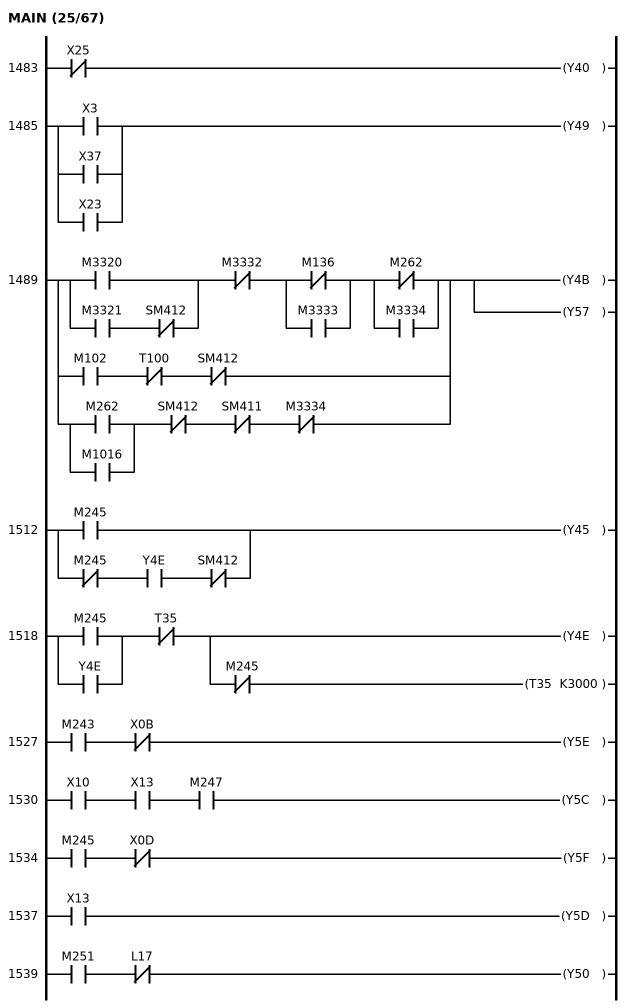
[picture p24: ladder of MAIN, rungs at steps 1483 to 1539]
1483  LDI     X25
      OUT     Y40
1485  LD      X3
      OR      X37
      OR      X23
      OUT     Y49
1489  LD      M3320
      LD      M3321
      ANI     SM412
      ORB
      ANI     M3332
      LDI     M136
      OR      M3333
      ANB
      LDI     M262
      OR      M3334
      ANB
      LD      M102
      ANI     T100
      ANI     SM412
      ORB
      LD      M262
      OR      M1016
      ANI     SM412
      ANI     SM411
      ANI     M3334
      ORB
      OUT     Y4B
      OUT     Y57
1512  LD      M245
      LDI     M245
      AND     Y4E
      ANI     SM412
      ORB
      OUT     Y45
1518  LD      M245
      OR      Y4E
      ANI     T35
      OUT     Y4E
      ANI     M245
      OUT     T35 K3000
1527  LD      M243
      ANI     X0B
      OUT     Y5E
1530  LD      X10
      AND     X13
      AND     M247
      OUT     Y5C
1534  LD      M245
      ANI     X0D
      OUT     Y5F
1537  LD      X13
      OUT     Y5D
1539  LD      M251
      ANI     L17
      OUT     Y50
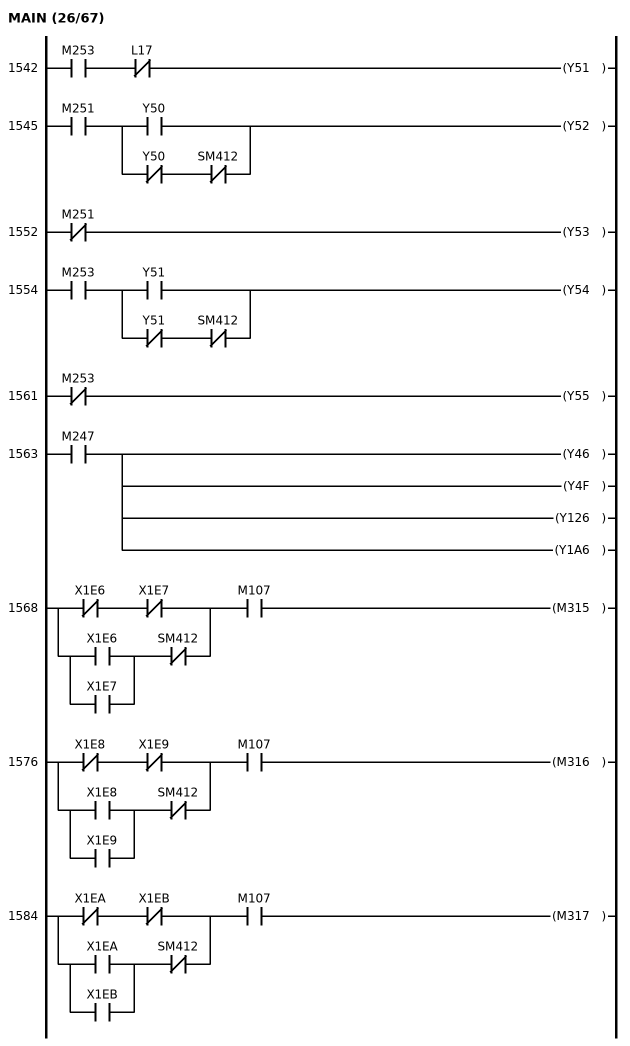
1542  LD      M253
      ANI     L17
      OUT     Y51
1545  LD      M251
      LD      Y50
      LDI     Y50
      ANI     SM412
      ORB
      ANB
      OUT     Y52
1552  LDI     M251
      OUT     Y53
1554  LD      M253
      LD      Y51
      LDI     Y51
      ANI     SM412
      ORB
      ANB
      OUT     Y54
1561  LDI     M253
      OUT     Y55
1563  LD      M247
      OUT     Y46
      OUT     Y4F
      OUT     Y126
      OUT     Y1A6
1568  LDI     X1E6
      ANI     X1E7
      LD      X1E6
      OR      X1E7
      ANI     SM412
      ORB
      AND     M107
      OUT     M315
1576  LDI     X1E8
      ANI     X1E9
      LD      X1E8
      OR      X1E9
      ANI     SM412
      ORB
      AND     M107
      OUT     M316
1584  LDI     X1EA
      ANI     X1EB
      LD      X1EA
      OR      X1EB
      ANI     SM412
      ORB
      AND     M107
      OUT     M317
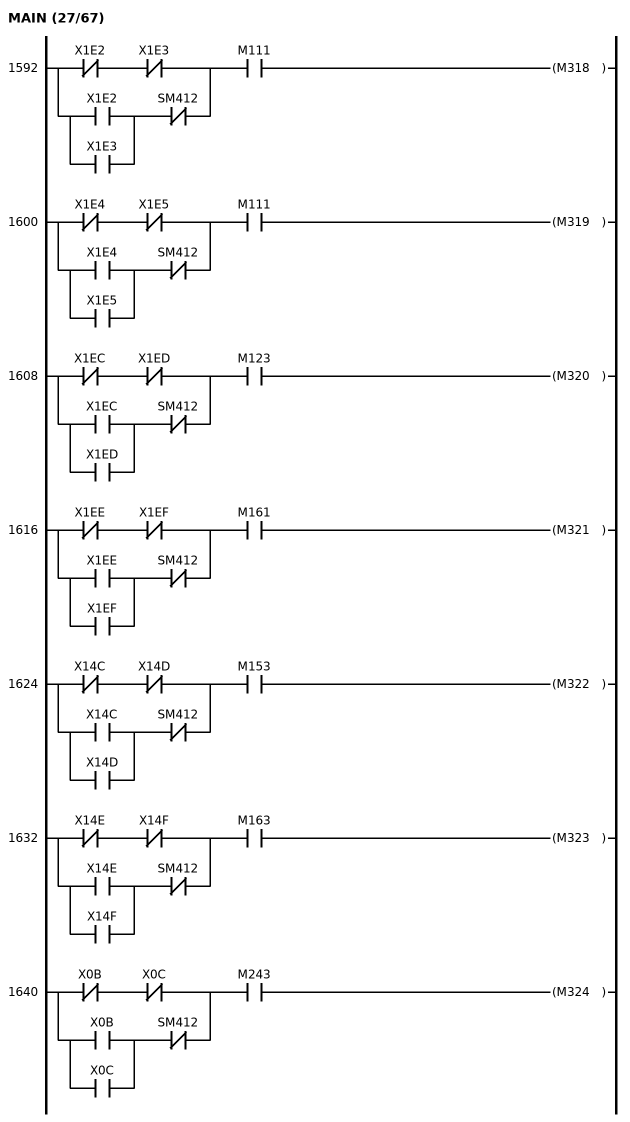
1592  LDI     X1E2
      ANI     X1E3
      LD      X1E2
      OR      X1E3
      ANI     SM412
      ORB
      AND     M111
      OUT     M318
1600  LDI     X1E4
      ANI     X1E5
      LD      X1E4
      OR      X1E5
      ANI     SM412
      ORB
      AND     M111
      OUT     M319
1608  LDI     X1EC
      ANI     X1ED
      LD      X1EC
      OR      X1ED
      ANI     SM412
      ORB
      AND     M123
      OUT     M320
1616  LDI     X1EE
      ANI     X1EF
      LD      X1EE
      OR      X1EF
      ANI     SM412
      ORB
      AND     M161
      OUT     M321
1624  LDI     X14C
      ANI     X14D
      LD      X14C
      OR      X14D
      ANI     SM412
      ORB
      AND     M153
      OUT     M322
1632  LDI     X14E
      ANI     X14F
      LD      X14E
      OR      X14F
      ANI     SM412
      ORB
      AND     M163
      OUT     M323
1640  LDI     X0B
      ANI     X0C
      LD      X0B
      OR      X0C
      ANI     SM412
      ORB
      AND     M243
      OUT     M324
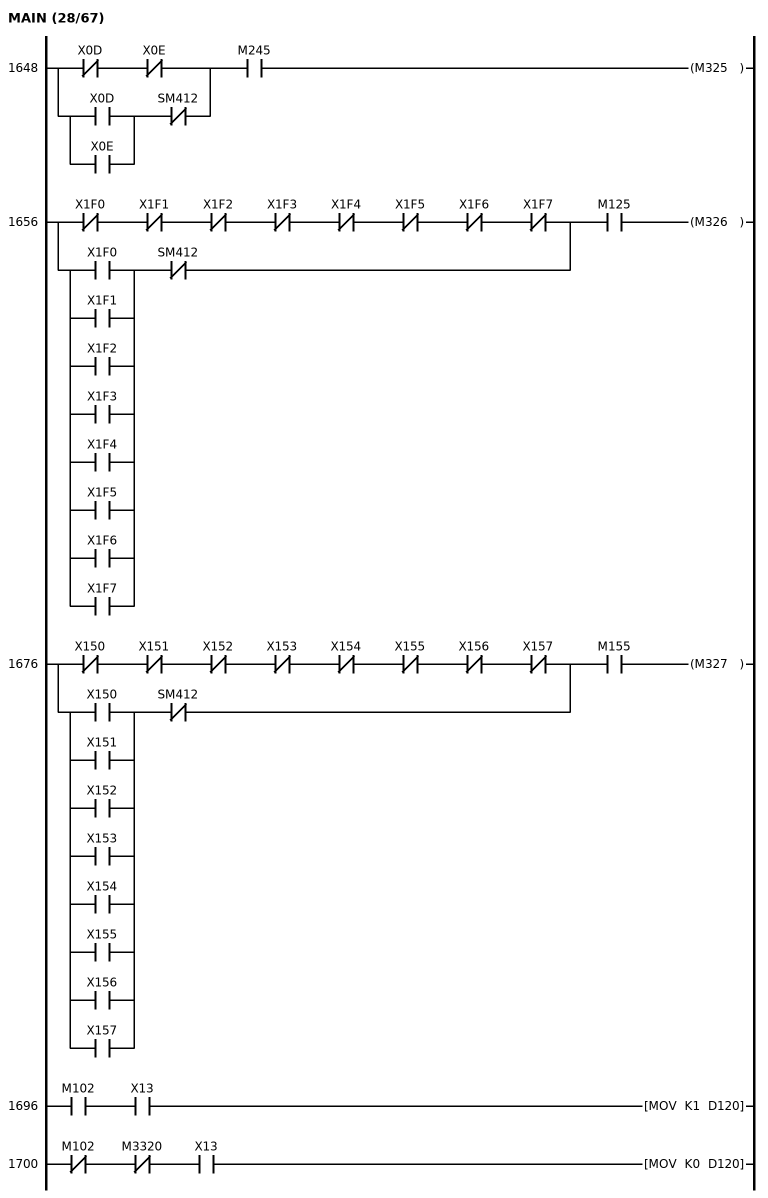
1648  LDI     X0D
      ANI     X0E
      LD      X0D
      OR      X0E
      ANI     SM412
      ORB
      AND     M245
      OUT     M325
1656  LDI     X1F0
      ANI     X1F1
      ANI     X1F2
      ANI     X1F3
      ANI     X1F4
      ANI     X1F5
      ANI     X1F6
      ANI     X1F7
      LD      X1F0
      OR      X1F1
      OR      X1F2
      OR      X1F3
      OR      X1F4
      OR      X1F5
      OR      X1F6
      OR      X1F7
      ANI     SM412
      ORB
      AND     M125
      OUT     M326
1676  LDI     X150
      ANI     X151
      ANI     X152
      ANI     X153
      ANI     X154
      ANI     X155
      ANI     X156
      ANI     X157
      LD      X150
      OR      X151
      OR      X152
      OR      X153
      OR      X154
      OR      X155
      OR      X156
      OR      X157
      ANI     SM412
      ORB
      AND     M155
      OUT     M327
1696  LD      M102
      AND     X13
      MOV     K1 D120
1700  LDI     M102
      ANI     M3320
      AND     X13
      MOV     K0 D120
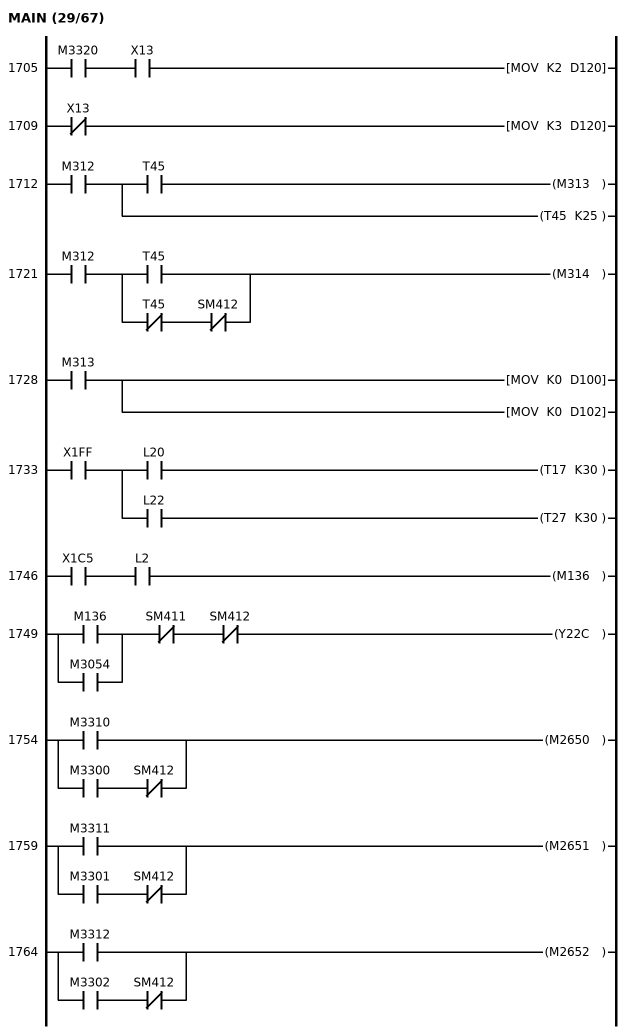
1705  LD      M3320
      AND     X13
      MOV     K2 D120
1709  LDI     X13
      MOV     K3 D120
1712  LD      M312
      MPS
      AND     T45
      OUT     M313
      MPP
      OUT     T45 K25
1721  LD      M312
      LD      T45
      LDI     T45
      ANI     SM412
      ORB
      ANB
      OUT     M314
1728  LD      M313
      MOV     K0 D100
      MOV     K0 D102
1733  LD      X1FF
      MPS
      AND     L20
      OUT     T17 K30
      MPP
      AND     L22
      OUT     T27 K30
1746  LD      X1C5
      AND     L2
      OUT     M136
1749  LD      M136
      OR      M3054
      ANI     SM411
      ANI     SM412
      OUT     Y22C
1754  LD      M3310
      LD      M3300
      ANI     SM412
      ORB
      OUT     M2650
1759  LD      M3311
      LD      M3301
      ANI     SM412
      ORB
      OUT     M2651
1764  LD      M3312
      LD      M3302
      ANI     SM412
      ORB
      OUT     M2652
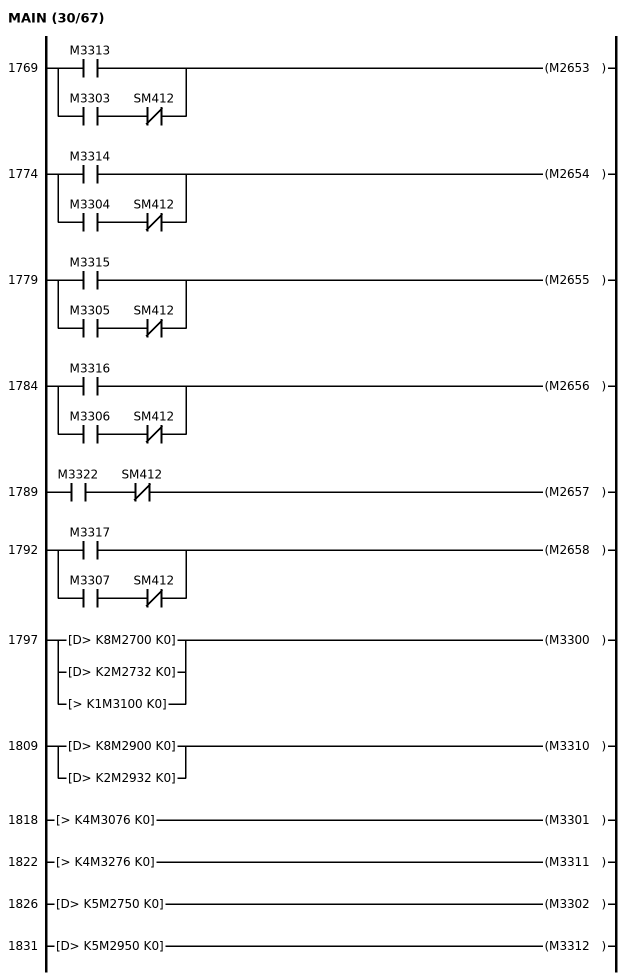
1769  LD      M3313
      LD      M3303
      ANI     SM412
      ORB
      OUT     M2653
1774  LD      M3314
      LD      M3304
      ANI     SM412
      ORB
      OUT     M2654
1779  LD      M3315
      LD      M3305
      ANI     SM412
      ORB
      OUT     M2655
1784  LD      M3316
      LD      M3306
      ANI     SM412
      ORB
      OUT     M2656
1789  LD      M3322
      ANI     SM412
      OUT     M2657
1792  LD      M3317
      LD      M3307
      ANI     SM412
      ORB
      OUT     M2658
1797  LDD>    K8M2700 K0
      ORD>    K2M2732 K0
      OR>     K1M3100 K0
      OUT     M3300
1809  LDD>    K8M2900 K0
      ORD>    K2M2932 K0
      OUT     M3310
1818  LD>     K4M3076 K0
      OUT     M3301
1822  LD>     K4M3276 K0
      OUT     M3311
1826  LDD>    K5M2750 K0
      OUT     M3302
1831  LDD>    K5M2950 K0
      OUT     M3312
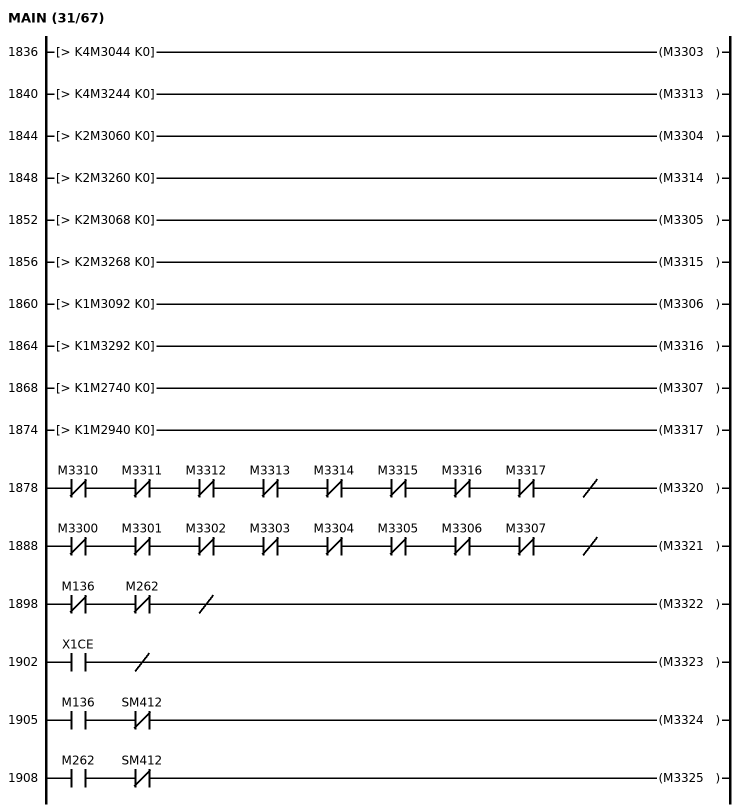
1836  LD>     K4M3044 K0
      OUT     M3303
1840  LD>     K4M3244 K0
      OUT     M3313
1844  LD>     K2M3060 K0
      OUT     M3304
1848  LD>     K2M3260 K0
      OUT     M3314
1852  LD>     K2M3068 K0
      OUT     M3305
1856  LD>     K2M3268 K0
      OUT     M3315
1860  LD>     K1M3092 K0
      OUT     M3306
1864  LD>     K1M3292 K0
      OUT     M3316
1868  LD>     K1M2740 K0
      OUT     M3307
        [note] 
1874  LD>     K1M2940 K0
      OUT     M3317
1878  LDI     M3310
      ANI     M3311
      ANI     M3312
      ANI     M3313
      ANI     M3314
      ANI     M3315
      ANI     M3316
      ANI     M3317
      INV
      OUT     M3320
1888  LDI     M3300
      ANI     M3301
      ANI     M3302
      ANI     M3303
      ANI     M3304
      ANI     M3305
      ANI     M3306
      ANI     M3307
      INV
      OUT     M3321
1898  LDI     M136
      ANI     M262
      INV
      OUT     M3322
1902  LD      X1CE
      INV
      OUT     M3323
1905  LD      M136
      ANI     SM412
      OUT     M3324
1908  LD      M262
      ANI     SM412
      OUT     M3325
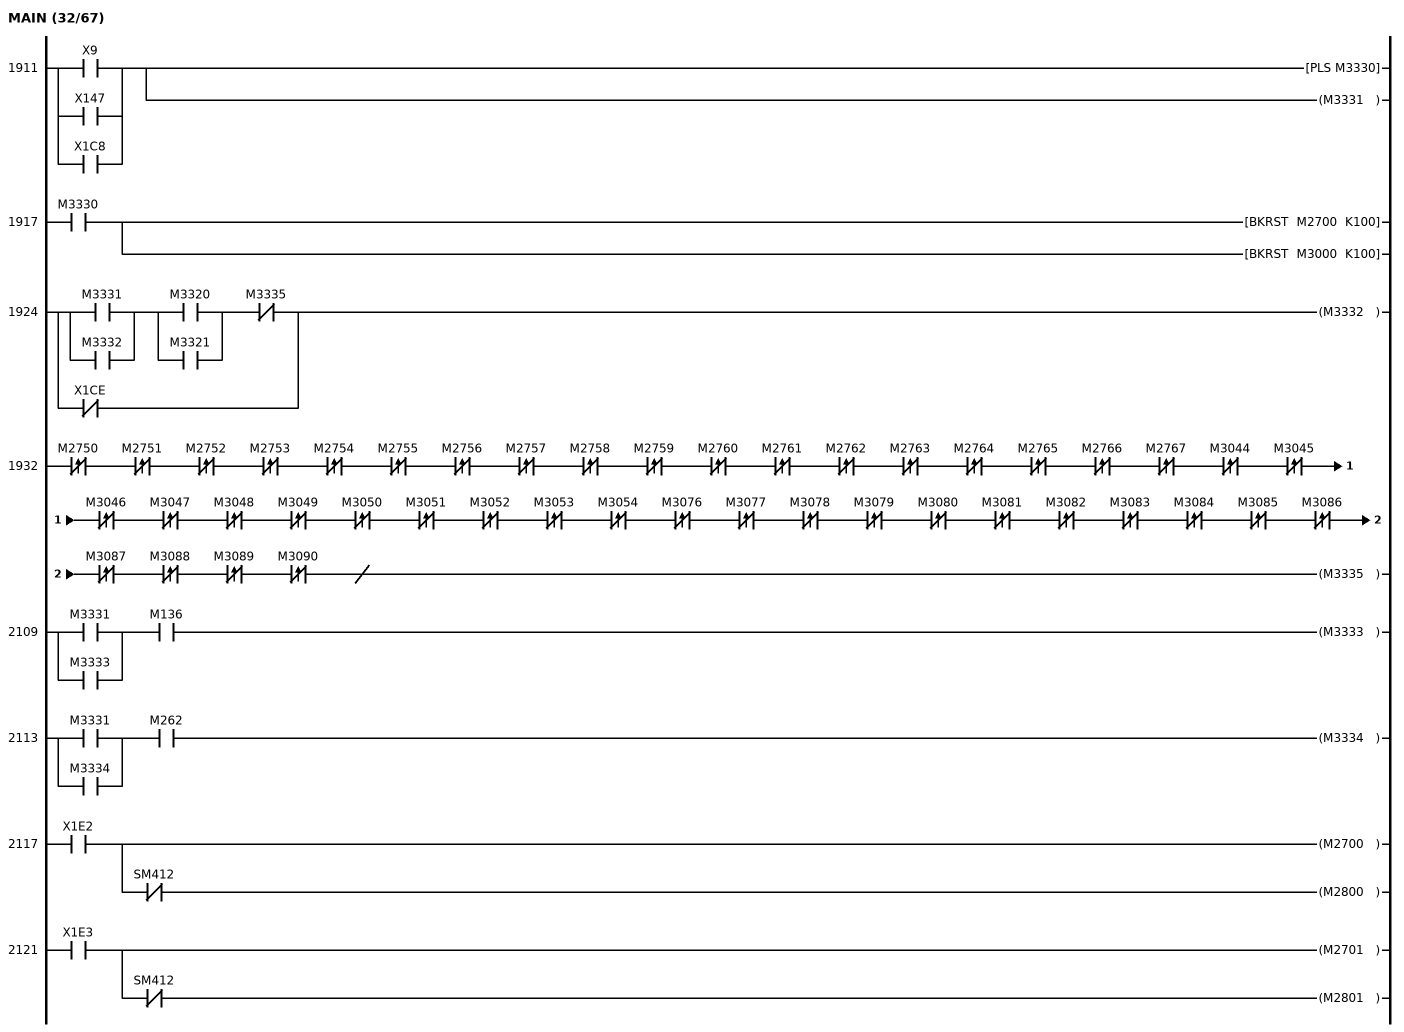
1911  LD      X9
      OR      X147
      OR      X1C8
      PLS     M3330
      OUT     M3331
1917  LD      M3330
      BKRST   M2700 K100
      BKRST   M3000 K100
1924  LD      M3331
      OR      M3332
      LD      M3320
      OR      M3321
      ANB
      ANI     M3335
      ORI     X1CE
      OUT     M3332
1932  LDPI    M2750
      ANDPI   M2751
      ANDPI   M2752
      ANDPI   M2753
      ANDPI   M2754
      ANDPI   M2755
      ANDPI   M2756
      ANDPI   M2757
      ANDPI   M2758
      ANDPI   M2759
      ANDPI   M2760
      ANDPI   M2761
      ANDPI   M2762
      ANDPI   M2763
      ANDPI   M2764
      ANDPI   M2765
      ANDPI   M2766
      ANDPI   M2767
      ANDPI   M3044
      ANDPI   M3045
      ANDPI   M3046
      ANDPI   M3047
      ANDPI   M3048
      ANDPI   M3049
      ANDPI   M3050
      ANDPI   M3051
      ANDPI   M3052
      ANDPI   M3053
      ANDPI   M3054
      ANDPI   M3076
      ANDPI   M3077
      ANDPI   M3078
      ANDPI   M3079
      ANDPI   M3080
      ANDPI   M3081
      ANDPI   M3082
      ANDPI   M3083
      ANDPI   M3084
      ANDPI   M3085
      ANDPI   M3086
      ANDPI   M3087
      ANDPI   M3088
      ANDPI   M3089
      ANDPI   M3090
      INV
      OUT     M3335
2109  LD      M3331
      OR      M3333
      AND     M136
      OUT     M3333
2113  LD      M3331
      OR      M3334
      AND     M262
      OUT     M3334
2117  LD      X1E2
      OUT     M2700
      ANI     SM412
      OUT     M2800
2121  LD      X1E3
      OUT     M2701
      ANI     SM412
      OUT     M2801
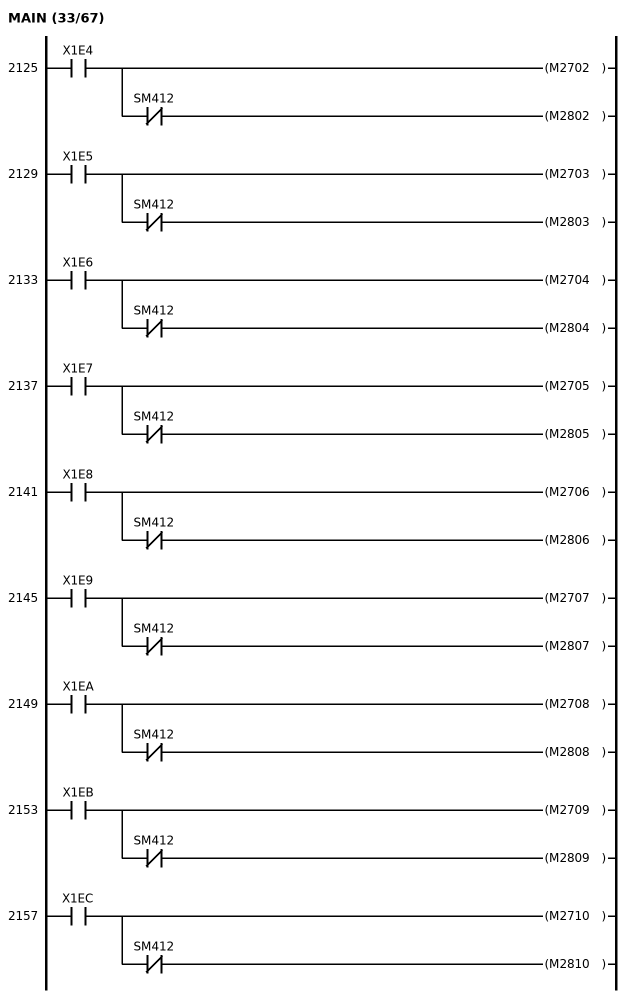
2125  LD      X1E4
      OUT     M2702
      ANI     SM412
      OUT     M2802
2129  LD      X1E5
      OUT     M2703
      ANI     SM412
      OUT     M2803
2133  LD      X1E6
      OUT     M2704
      ANI     SM412
      OUT     M2804
2137  LD      X1E7
      OUT     M2705
      ANI     SM412
      OUT     M2805
2141  LD      X1E8
      OUT     M2706
      ANI     SM412
      OUT     M2806
2145  LD      X1E9
      OUT     M2707
      ANI     SM412
      OUT     M2807
2149  LD      X1EA
      OUT     M2708
      ANI     SM412
      OUT     M2808
2153  LD      X1EB
      OUT     M2709
      ANI     SM412
      OUT     M2809
2157  LD      X1EC
      OUT     M2710
      ANI     SM412
      OUT     M2810
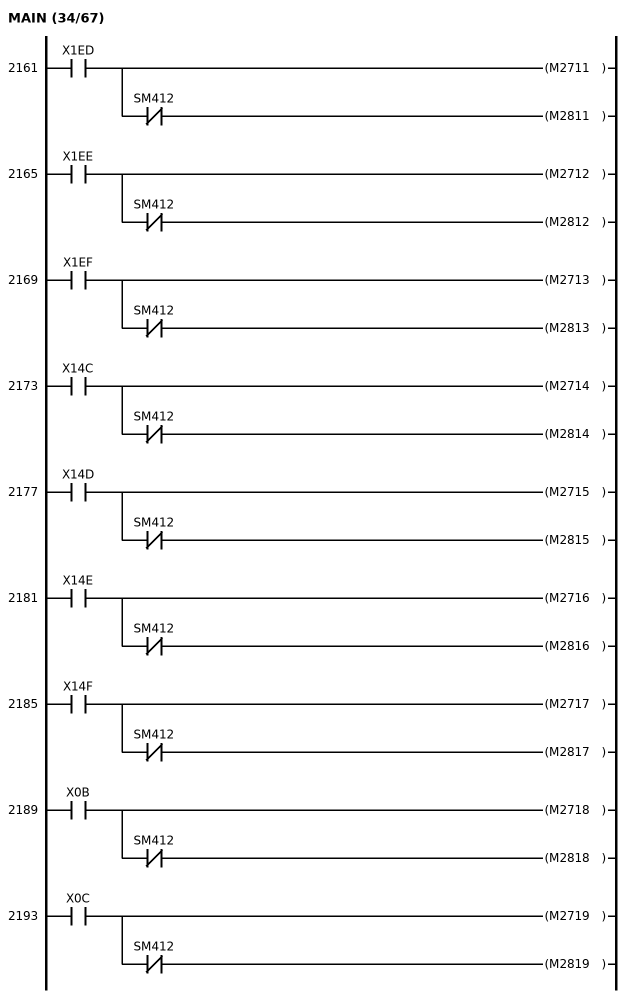
2161  LD      X1ED
      OUT     M2711
      ANI     SM412
      OUT     M2811
2165  LD      X1EE
      OUT     M2712
      ANI     SM412
      OUT     M2812
2169  LD      X1EF
      OUT     M2713
      ANI     SM412
      OUT     M2813
2173  LD      X14C
      OUT     M2714
      ANI     SM412
      OUT     M2814
2177  LD      X14D
      OUT     M2715
      ANI     SM412
      OUT     M2815
2181  LD      X14E
      OUT     M2716
      ANI     SM412
      OUT     M2816
2185  LD      X14F
      OUT     M2717
      ANI     SM412
      OUT     M2817
2189  LD      X0B
      OUT     M2718
      ANI     SM412
      OUT     M2818
2193  LD      X0C
      OUT     M2719
      ANI     SM412
      OUT     M2819
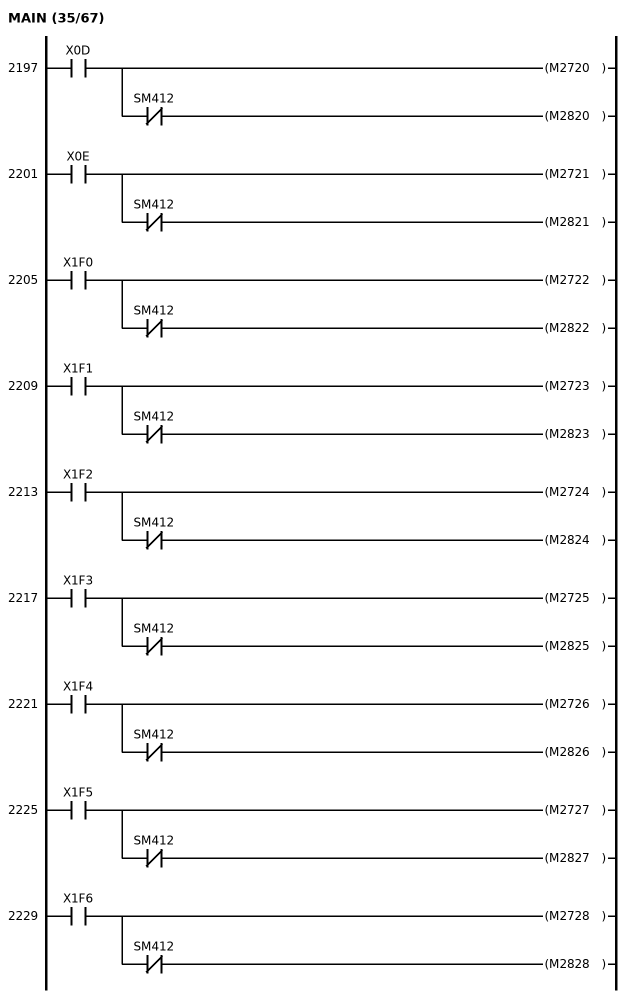
2197  LD      X0D
      OUT     M2720
      ANI     SM412
      OUT     M2820
2201  LD      X0E
      OUT     M2721
      ANI     SM412
      OUT     M2821
2205  LD      X1F0
      OUT     M2722
      ANI     SM412
      OUT     M2822
2209  LD      X1F1
      OUT     M2723
      ANI     SM412
      OUT     M2823
2213  LD      X1F2
      OUT     M2724
      ANI     SM412
      OUT     M2824
2217  LD      X1F3
      OUT     M2725
      ANI     SM412
      OUT     M2825
2221  LD      X1F4
      OUT     M2726
      ANI     SM412
      OUT     M2826
2225  LD      X1F5
      OUT     M2727
      ANI     SM412
      OUT     M2827
2229  LD      X1F6
      OUT     M2728
      ANI     SM412
      OUT     M2828
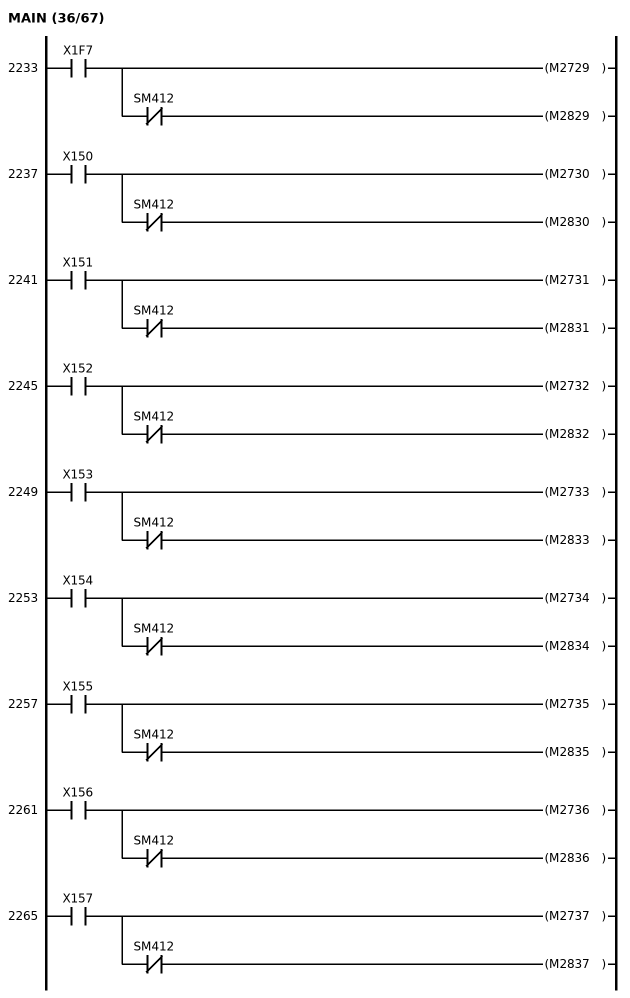
2233  LD      X1F7
      OUT     M2729
      ANI     SM412
      OUT     M2829
2237  LD      X150
      OUT     M2730
      ANI     SM412
      OUT     M2830
2241  LD      X151
      OUT     M2731
      ANI     SM412
      OUT     M2831
2245  LD      X152
      OUT     M2732
      ANI     SM412
      OUT     M2832
2249  LD      X153
      OUT     M2733
      ANI     SM412
      OUT     M2833
2253  LD      X154
      OUT     M2734
      ANI     SM412
      OUT     M2834
2257  LD      X155
      OUT     M2735
      ANI     SM412
      OUT     M2835
2261  LD      X156
      OUT     M2736
      ANI     SM412
      OUT     M2836
2265  LD      X157
      OUT     M2737
      ANI     SM412
      OUT     M2837
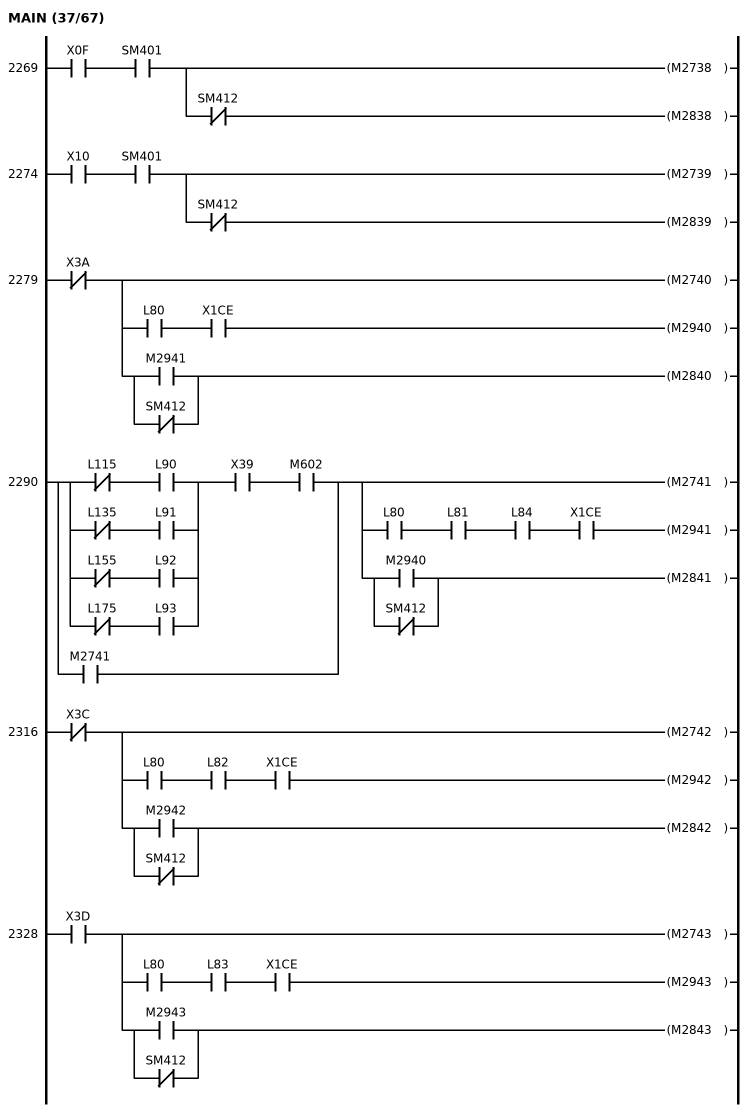
2269  LD      X0F
      AND     SM401
      OUT     M2738
      ANI     SM412
      OUT     M2838
2274  LD      X10
      AND     SM401
      OUT     M2739
      ANI     SM412
      OUT     M2839
2279  LDI     X3A
      OUT     M2740
      MPS
      AND     L80
      AND     X1CE
      OUT     M2940
      MPP
      LD      M2941
      ORI     SM412
      ANB
      OUT     M2840
2290  LDI     L115
      AND     L90
      LDI     L135
      AND     L91
      ORB
      LDI     L155
      AND     L92
      ORB
      LDI     L175
      AND     L93
      ORB
      AND     X39
      AND     M602
      OR      M2741
      OUT     M2741
      MPS
      AND     L80
      AND     L81
      AND     L84
      AND     X1CE
      OUT     M2941
      MPP
      LD      M2940
      ORI     SM412
      ANB
      OUT     M2841
2316  LDI     X3C
      OUT     M2742
      MPS
      AND     L80
      AND     L82
      AND     X1CE
      OUT     M2942
      MPP
      LD      M2942
      ORI     SM412
      ANB
      OUT     M2842
2328  LD      X3D
      OUT     M2743
      MPS
      AND     L80
      AND     L83
      AND     X1CE
      OUT     M2943
      MPP
      LD      M2943
      ORI     SM412
      ANB
      OUT     M2843
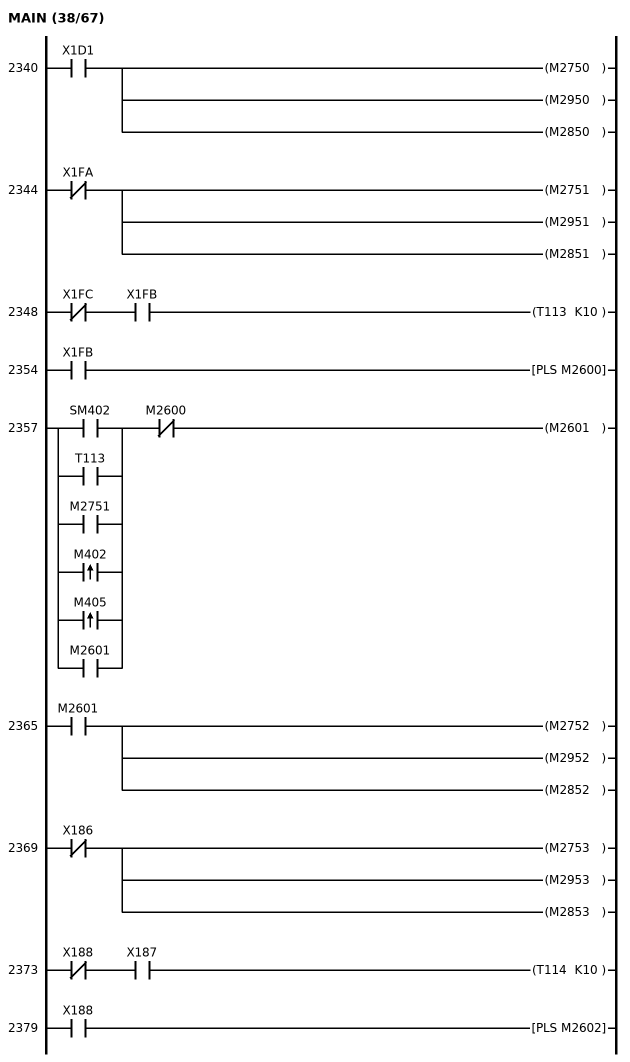
2340  LD      X1D1
      OUT     M2750
      OUT     M2950
      OUT     M2850
2344  LDI     X1FA
      OUT     M2751
      OUT     M2951
      OUT     M2851
2348  LDI     X1FC
      AND     X1FB
      OUT     T113 K10
2354  LD      X1FB
      PLS     M2600
2357  LD      SM402
      OR      T113
      OR      M2751
      ORP     M402
      ORP     M405
      OR      M2601
      ANI     M2600
      OUT     M2601
2365  LD      M2601
      OUT     M2752
      OUT     M2952
      OUT     M2852
2369  LDI     X186
      OUT     M2753
      OUT     M2953
      OUT     M2853
2373  LDI     X188
      AND     X187
      OUT     T114 K10
2379  LD      X188
      PLS     M2602
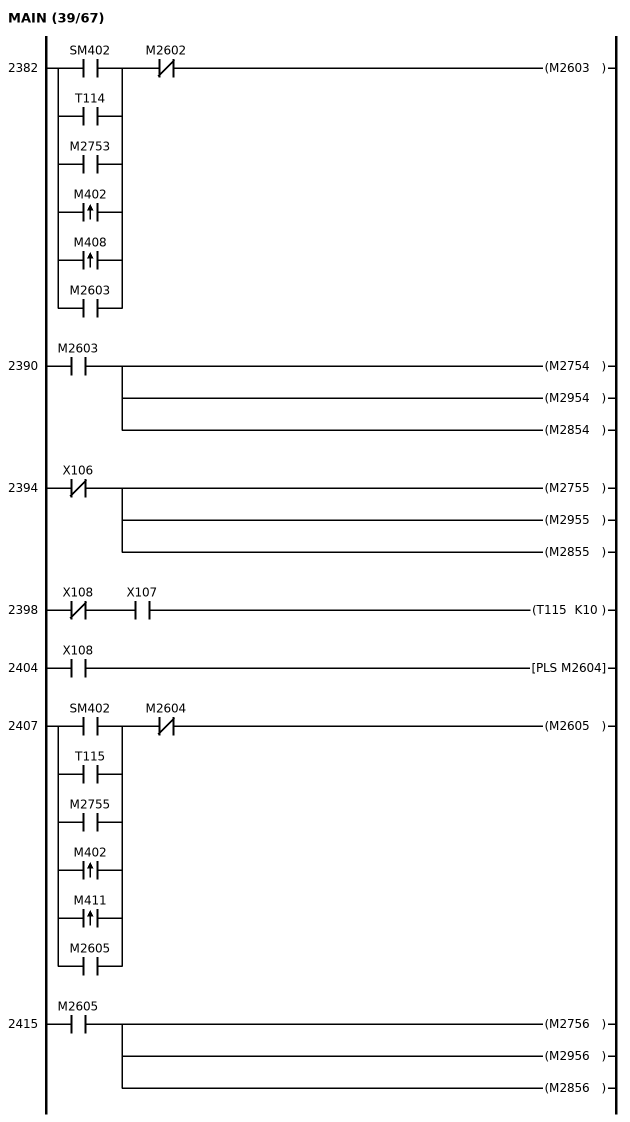
2382  LD      SM402
      OR      T114
      OR      M2753
      ORP     M402
      ORP     M408
      OR      M2603
      ANI     M2602
      OUT     M2603
2390  LD      M2603
      OUT     M2754
      OUT     M2954
      OUT     M2854
2394  LDI     X106
      OUT     M2755
      OUT     M2955
      OUT     M2855
2398  LDI     X108
      AND     X107
      OUT     T115 K10
2404  LD      X108
      PLS     M2604
2407  LD      SM402
      OR      T115
      OR      M2755
      ORP     M402
      ORP     M411
      OR      M2605
      ANI     M2604
      OUT     M2605
2415  LD      M2605
      OUT     M2756
      OUT     M2956
      OUT     M2856
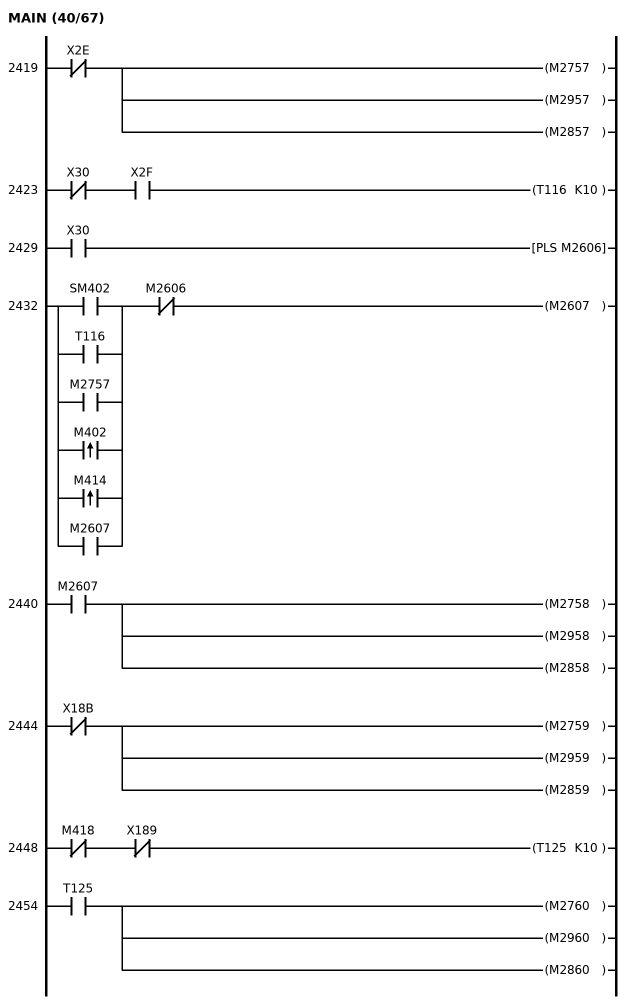
2419  LDI     X2E
      OUT     M2757
      OUT     M2957
      OUT     M2857
2423  LDI     X30
      AND     X2F
      OUT     T116 K10
2429  LD      X30
      PLS     M2606
2432  LD      SM402
      OR      T116
      OR      M2757
      ORP     M402
      ORP     M414
      OR      M2607
      ANI     M2606
      OUT     M2607
2440  LD      M2607
      OUT     M2758
      OUT     M2958
      OUT     M2858
2444  LDI     X18B
      OUT     M2759
      OUT     M2959
      OUT     M2859
2448  LDI     M418
      ANI     X189
      OUT     T125 K10
2454  LD      T125
      OUT     M2760
      OUT     M2960
      OUT     M2860
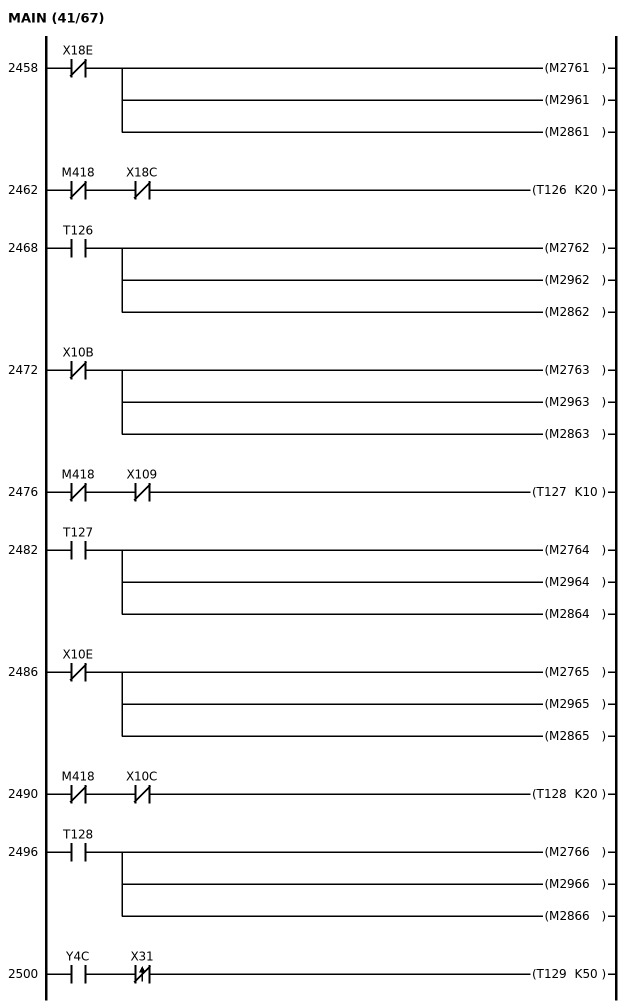
2458  LDI     X18E
      OUT     M2761
      OUT     M2961
      OUT     M2861
2462  LDI     M418
      ANI     X18C
      OUT     T126 K20
2468  LD      T126
      OUT     M2762
      OUT     M2962
      OUT     M2862
2472  LDI     X10B
      OUT     M2763
      OUT     M2963
      OUT     M2863
2476  LDI     M418
      ANI     X109
      OUT     T127 K10
2482  LD      T127
      OUT     M2764
      OUT     M2964
      OUT     M2864
2486  LDI     X10E
      OUT     M2765
      OUT     M2965
      OUT     M2865
2490  LDI     M418
      ANI     X10C
      OUT     T128 K20
2496  LD      T128
      OUT     M2766
      OUT     M2966
      OUT     M2866
2500  LD      Y4C
      ANDPI   X31
      OUT     T129 K50
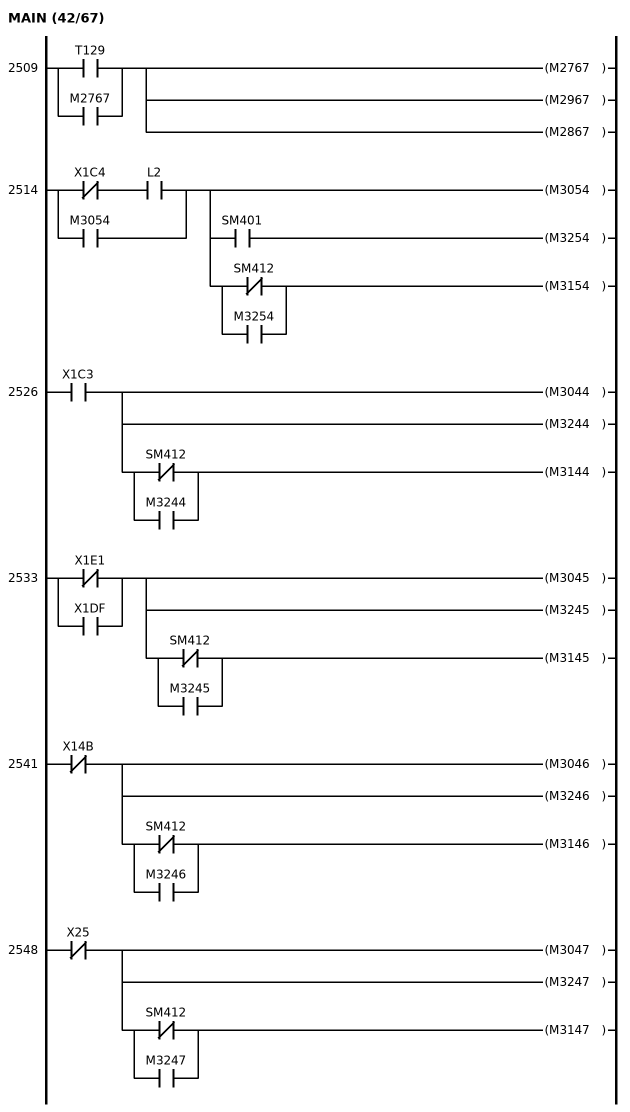
2509  LD      T129
      OR      M2767
      OUT     M2767
      OUT     M2967
      OUT     M2867
2514  LDI     X1C4
      AND     L2
      OR      M3054
      OUT     M3054
      MPS
      AND     SM401
      OUT     M3254
      MPP
      LDI     SM412
      OR      M3254
      ANB
      OUT     M3154
2526  LD      X1C3
      OUT     M3044
      OUT     M3244
      LDI     SM412
      OR      M3244
      ANB
      OUT     M3144
2533  LDI     X1E1
      OR      X1DF
      OUT     M3045
      OUT     M3245
      LDI     SM412
      OR      M3245
      ANB
      OUT     M3145
2541  LDI     X14B
      OUT     M3046
      OUT     M3246
      LDI     SM412
      OR      M3246
      ANB
      OUT     M3146
2548  LDI     X25
      OUT     M3047
      OUT     M3247
      LDI     SM412
      OR      M3247
      ANB
      OUT     M3147
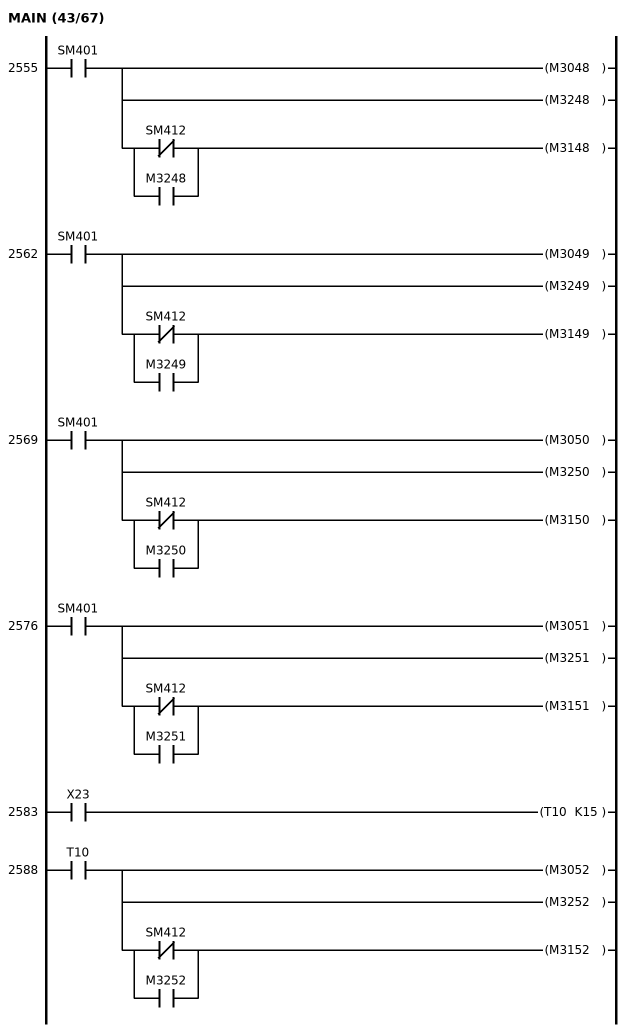
2555  LD      SM401
      OUT     M3048
      OUT     M3248
      LDI     SM412
      OR      M3248
      ANB
      OUT     M3148
2562  LD      SM401
      OUT     M3049
      OUT     M3249
      LDI     SM412
      OR      M3249
      ANB
      OUT     M3149
2569  LD      SM401
      OUT     M3050
      OUT     M3250
      LDI     SM412
      OR      M3250
      ANB
      OUT     M3150
2576  LD      SM401
      OUT     M3051
      OUT     M3251
      LDI     SM412
      OR      M3251
      ANB
      OUT     M3151
2583  LD      X23
      OUT     T10 K15
2588  LD      T10
      OUT     M3052
      OUT     M3252
      LDI     SM412
      OR      M3252
      ANB
      OUT     M3152
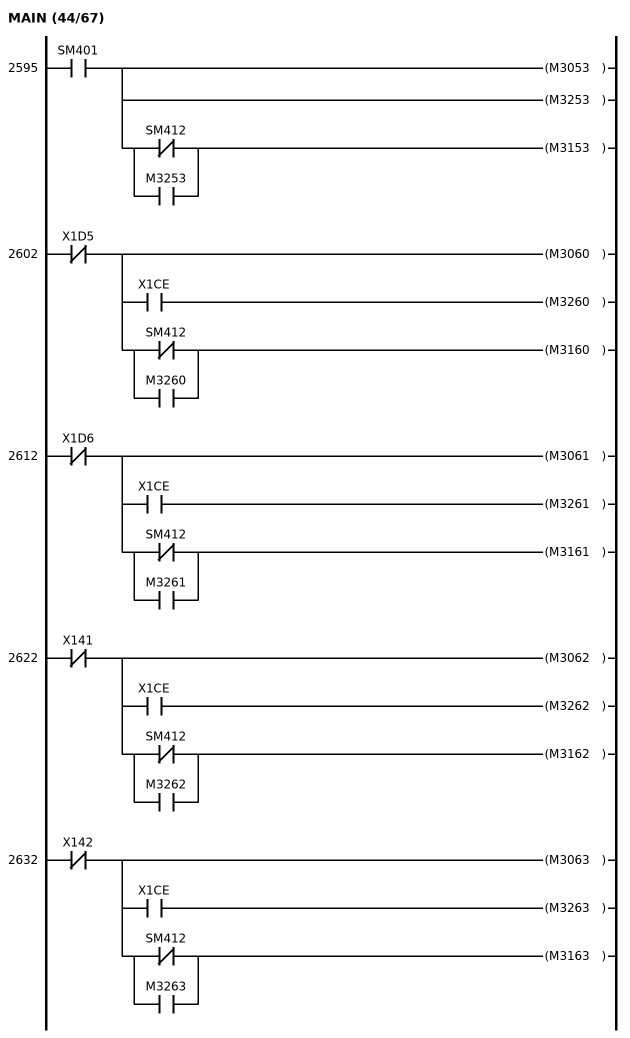
2595  LD      SM401
      OUT     M3053
      OUT     M3253
      LDI     SM412
      OR      M3253
      ANB
      OUT     M3153
2602  LDI     X1D5
      OUT     M3060
      MPS
      AND     X1CE
      OUT     M3260
      MPP
      LDI     SM412
      OR      M3260
      ANB
      OUT     M3160
2612  LDI     X1D6
      OUT     M3061
      MPS
      AND     X1CE
      OUT     M3261
      MPP
      LDI     SM412
      OR      M3261
      ANB
      OUT     M3161
2622  LDI     X141
      OUT     M3062
      MPS
      AND     X1CE
      OUT     M3262
      MPP
      LDI     SM412
      OR      M3262
      ANB
      OUT     M3162
2632  LDI     X142
      OUT     M3063
      MPS
      AND     X1CE
      OUT     M3263
      MPP
      LDI     SM412
      OR      M3263
      ANB
      OUT     M3163
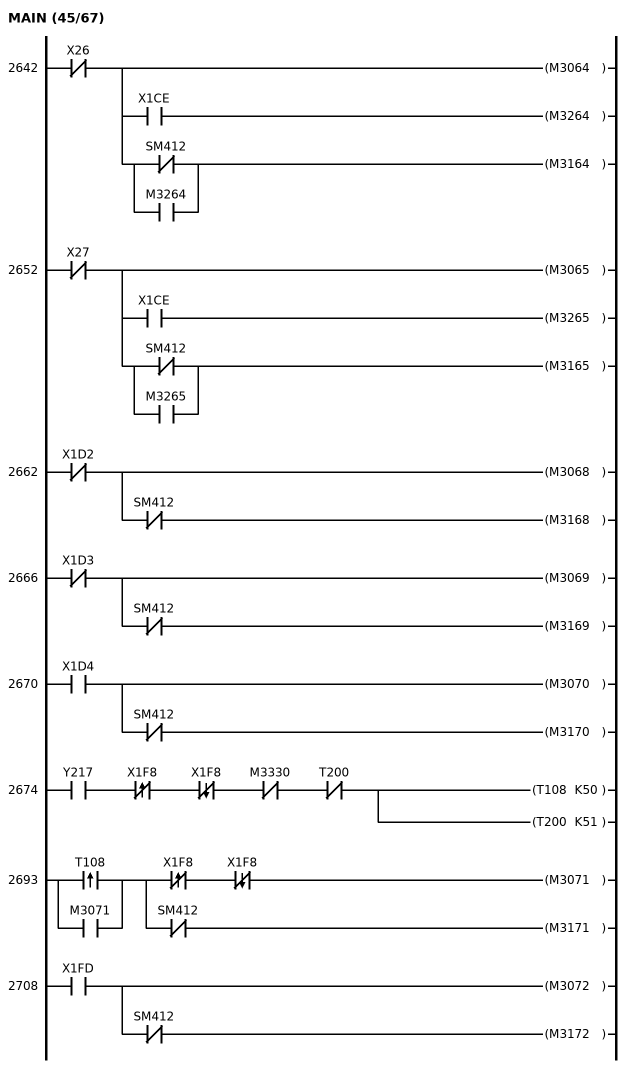
2642  LDI     X26
      OUT     M3064
      MPS
      AND     X1CE
      OUT     M3264
      MPP
      LDI     SM412
      OR      M3264
      ANB
      OUT     M3164
2652  LDI     X27
      OUT     M3065
      MPS
      AND     X1CE
      OUT     M3265
      MPP
      LDI     SM412
      OR      M3265
      ANB
      OUT     M3165
2662  LDI     X1D2
      OUT     M3068
      ANI     SM412
      OUT     M3168
2666  LDI     X1D3
      OUT     M3069
      ANI     SM412
      OUT     M3169
2670  LD      X1D4
      OUT     M3070
      ANI     SM412
      OUT     M3170
2674  LD      Y217
      ANDPI   X1F8
      ANDFI   X1F8
      ANI     M3330
      ANI     T200
      OUT     T108 K50
      OUT     T200 K51
2693  LDP     T108
      OR      M3071
      MPS
      ANDPI   X1F8
      ANDFI   X1F8
      OUT     M3071
      MPP
      ANI     SM412
      OUT     M3171
2708  LD      X1FD
      OUT     M3072
      ANI     SM412
      OUT     M3172
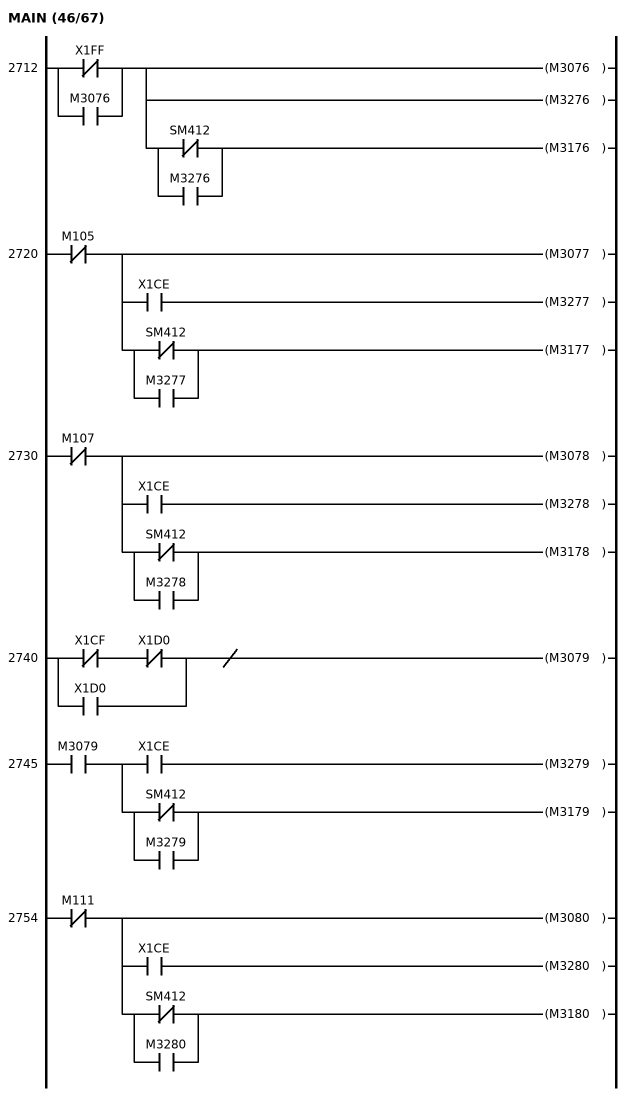
2712  LDI     X1FF
      OR      M3076
      OUT     M3076
      OUT     M3276
      LDI     SM412
      OR      M3276
      ANB
      OUT     M3176
2720  LDI     M105
      OUT     M3077
      MPS
      AND     X1CE
      OUT     M3277
      MPP
      LDI     SM412
      OR      M3277
      ANB
      OUT     M3177
2730  LDI     M107
      OUT     M3078
      MPS
      AND     X1CE
      OUT     M3278
      MPP
      LDI     SM412
      OR      M3278
      ANB
      OUT     M3178
2740  LDI     X1CF
      ANI     X1D0
      OR      X1D0
      INV
      OUT     M3079
2745  LD      M3079
      MPS
      AND     X1CE
      OUT     M3279
      MPP
      LDI     SM412
      OR      M3279
      ANB
      OUT     M3179
2754  LDI     M111
      OUT     M3080
      MPS
      AND     X1CE
      OUT     M3280
      MPP
      LDI     SM412
      OR      M3280
      ANB
      OUT     M3180
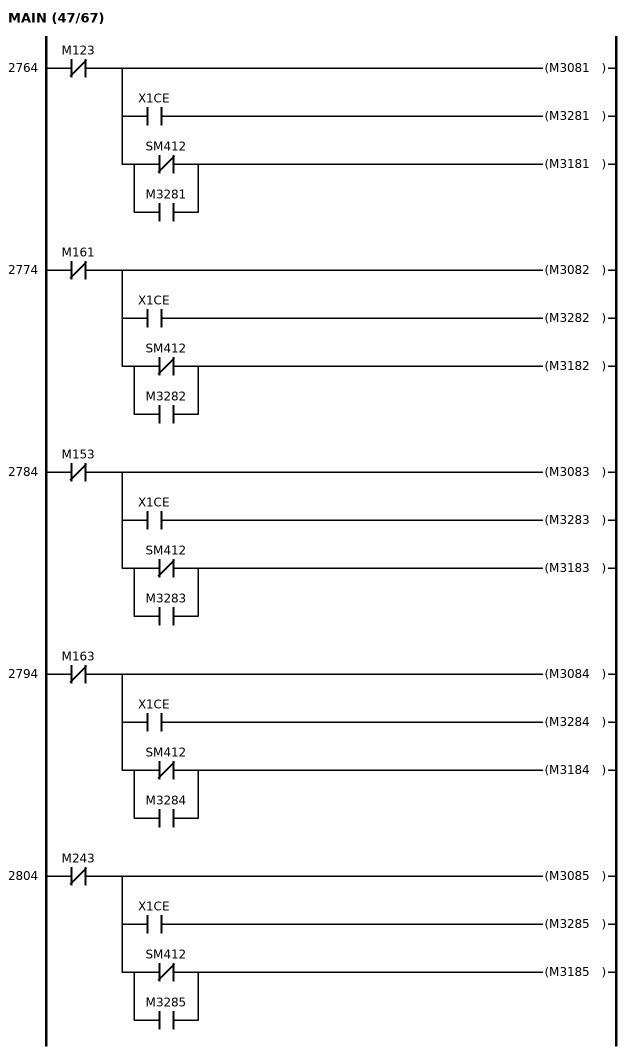
2764  LDI     M123
      OUT     M3081
      MPS
      AND     X1CE
      OUT     M3281
      MPP
      LDI     SM412
      OR      M3281
      ANB
      OUT     M3181
2774  LDI     M161
      OUT     M3082
      MPS
      AND     X1CE
      OUT     M3282
      MPP
      LDI     SM412
      OR      M3282
      ANB
      OUT     M3182
2784  LDI     M153
      OUT     M3083
      MPS
      AND     X1CE
      OUT     M3283
      MPP
      LDI     SM412
      OR      M3283
      ANB
      OUT     M3183
2794  LDI     M163
      OUT     M3084
      MPS
      AND     X1CE
      OUT     M3284
      MPP
      LDI     SM412
      OR      M3284
      ANB
      OUT     M3184
2804  LDI     M243
      OUT     M3085
      MPS
      AND     X1CE
      OUT     M3285
      MPP
      LDI     SM412
      OR      M3285
      ANB
      OUT     M3185
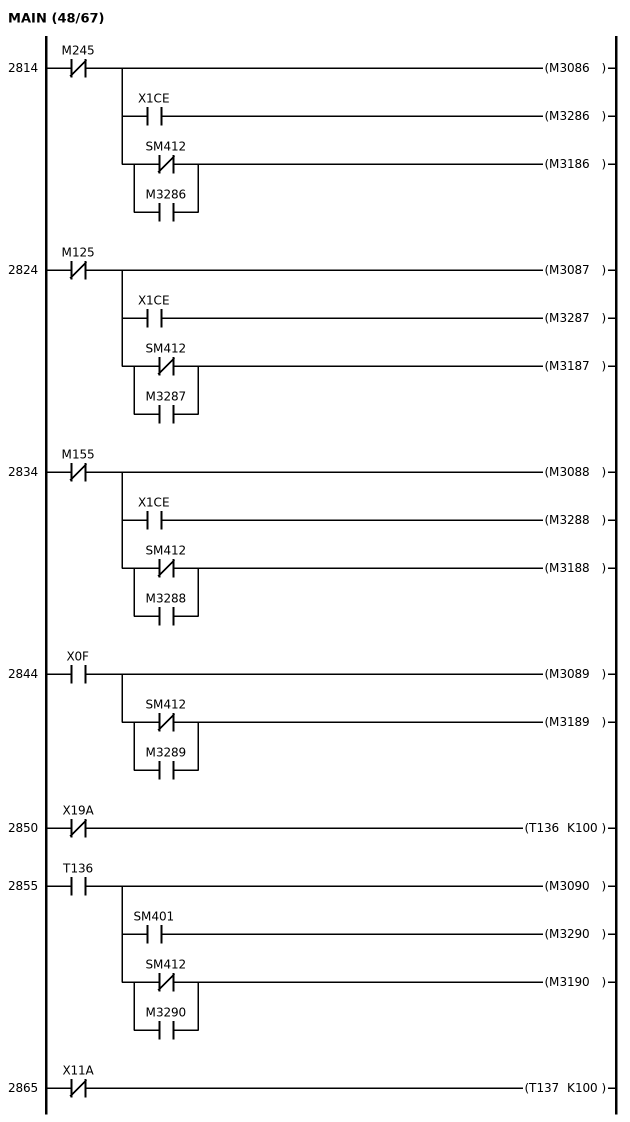
2814  LDI     M245
      OUT     M3086
      MPS
      AND     X1CE
      OUT     M3286
      MPP
      LDI     SM412
      OR      M3286
      ANB
      OUT     M3186
2824  LDI     M125
      OUT     M3087
      MPS
      AND     X1CE
      OUT     M3287
      MPP
      LDI     SM412
      OR      M3287
      ANB
      OUT     M3187
2834  LDI     M155
      OUT     M3088
      MPS
      AND     X1CE
      OUT     M3288
      MPP
      LDI     SM412
      OR      M3288
      ANB
      OUT     M3188
2844  LD      X0F
      OUT     M3089
      LDI     SM412
      OR      M3289
      ANB
      OUT     M3189
2850  LDI     X19A
      OUT     T136 K100
2855  LD      T136
      OUT     M3090
      MPS
      AND     SM401
      OUT     M3290
      MPP
      LDI     SM412
      OR      M3290
      ANB
      OUT     M3190
2865  LDI     X11A
      OUT     T137 K100
